# EPICS autosave request: iocBoot/iocEPU1/velocity.req
$(SYS){$(DEV)}-GapMtrSpd
$(SYS){$(DEV)}-PhaseMtrSpd
